// TwinCAT 3 PLC project Rajang
// ProgramVersion: 3.1.4024.0
// libraries:
//   Tc2_Standard, * (Beckhoff Automation GmbH)
//   Tc2_System, * (Beckhoff Automation GmbH)
//   Tc3_Module, * (Beckhoff Automation GmbH)
// project tree:
//   / PlcTask.TcTTO
//   POUs/ Lamp.TcPOU, Light.TcPOU, MAIN.TcPOU
// real-time tasks:
//   TASK PlcTask: cycle T#10ms, priority 20, ADS port 350
// motion (NC):
// I/O:
//   DEVICE Its1 (EtherCAT), AmsNetId 10.200.224.204.2.1
//     Term 1 (EK1100) [EK1100 EtherCAT Coupler (2A E-Bus)]
//       Term 3 (EL1002) [EL1002 2Ch. Dig. Input 24V, 3ms]
//       Term 4 (EL1004) [EL1004 4Ch. Dig. Input 24V, 3ms]
//     Drive 2 (AX5203-0000-0203) [AX5203-0000-0203 EtherCAT Drive (SoE, 2 Ch.)]

CONFIGURATION Rajang
    RESOURCE PLC ON TwinCAT3
        TASK PlcTask(INTERVAL := T#10ms, PRIORITY := 20);
        PROGRAM MAIN WITH PlcTask : MAIN;
    END_RESOURCE
END_CONFIGURATION

// ---- POUs/MAIN.TcPOU
PROGRAM MAIN
VAR
	input : BOOL;
	output : bool;
END_VAR

input := output;
Light();
Lamp();

END_PROGRAM

// ---- POUs/Light.TcPOU
PROGRAM Light
VAR
	Counter: int;
END_VAR

Counter := Counter +22;

END_PROGRAM

// ---- POUs/Lamp.TcPOU
PROGRAM Lamp
VAR
	countercounter : int;
END_VAR

countercounter := countercounter +1;

END_PROGRAM
